// Mitsubishi GX Works2 project: ProjectGroup11   PLC: FX3G

// global labels: Global1
VAR_GLOBAL
  StartSwitch AT X002 : BOOL;
  TC_1 AT TC1 : BOOL;
END_VAR
VAR_GLOBAL CONSTANT
  VALUE : INT := 30;
END_VAR
VAR_GLOBAL
  TS_1 AT TS1 : BOOL;
  Y_005 AT Y005 : BOOL;
  OrangeStock AT D1100 : REAL;
  ClementinesStock AT D1102 : REAL;
  PomeloStock : REAL;
  OrangeWash AT D1106 : REAL;
  ClementinesWash AT D1108 : REAL;
  PomeloWash AT D1110 : REAL;
  SquizeContainer AT D1112 : REAL;
END_VAR
VAR_GLOBAL CONSTANT
  MaxOrangeWash : REAL := 100;
END_VAR
VAR_GLOBAL
  collectionSwitch AT X001 : BOOL;
  collectionInProcess AT Y001 : BOOL;
  squizeSwitch AT X011 : BOOL;
  CC_11 AT CC11 : BOOL;
END_VAR
VAR_GLOBAL CONSTANT
  CS11 : INT := 2;
  const : INT := 2;
END_VAR
VAR_GLOBAL
  CS_11 AT CS11 : BOOL;
  StartDaySwitch AT X010 : BOOL;
END_VAR
VAR_GLOBAL CONSTANT
  MinOranges : REAL;
  PomelaCon : REAL;
  ClementinCon : REAL;
END_VAR
VAR_GLOBAL
  Y_10 AT Y010 : BOOL;
  OffSwitch AT X007 : BOOL;
  TC_7 AT TC7 : BOOL;
END_VAR
VAR_GLOBAL CONSTANT
  ValueOff : INT := 30;
  ValueStart1 : INT := 30;
END_VAR
VAR_GLOBAL
  Y_010 AT Y010 : BOOL;
  M_0 AT M0 : BOOL;
  X_7 AT X007 : BOOL;
  TC_200 AT TC200 : BOOL;
  M_1 AT M1 : BOOL;
  TC_2 AT TC2 : BOOL;
  TS_2 AT TS2 : BOOL;
  M_2 AT M2 : BOOL;
  firstBlink AT M3 : BOOL;
  TC_3 AT TC3 : BOOL;
END_VAR
VAR_GLOBAL CONSTANT
  BlinkingTime : INT := 5;
END_VAR
VAR_GLOBAL
  TS_3 AT TS3 : BOOL;
  Blink2 AT M4 : BOOL;
  Blink1 AT M3 : BOOL;
  TC_4 AT TC4 : BOOL;
  TS_4 AT TS4 : BOOL;
  Blink3 AT M5 : BOOL;
  AllGood AT M6 : BOOL;
  NotGood AT M6 : BOOL;
  StartWashSwitch AT X002 : BOOL;
  Wash1 AT M7 : BOOL;
END_VAR
VAR_GLOBAL CONSTANT
  Ratio : REAL := 2.0;
END_VAR
VAR_GLOBAL
  NumOfOrangeToWash AT D1114 : REAL;
  squize1 AT M8 : BOOL;
  fruitToSquize AT D1116 : REAL;
  switchon AT M1 : BOOL;
  MHelp AT X000 : BOOL;
  Help AT M40 : BOOL;
  Y_6 AT Y006 : BOOL;
  M_35 AT M35 : BOOL;
  JuiceTank AT D1118 : REAL;
  M_9 AT M9 : BOOL;
  TC_5 AT TC5 : BOOL;
END_VAR
VAR_GLOBAL CONSTANT
  SquizeTime : INT := 30;
END_VAR
VAR_GLOBAL
  TS_5 AT TS5 : BOOL;
  Y_2 AT Y002 : BOOL;
  Y_3 AT Y003 : BOOL;
  M_10 AT M10 : BOOL;
  CHECK_QUALIY_STAGE AT X003 : BOOL;
  Output AT D1120 : INT;
END_VAR
VAR_GLOBAL CONSTANT
  UpperBound : REAL := 5.0;
  LowerBound : REAL := 1.0;
END_VAR
VAR_GLOBAL
  M_11 AT M11 : BOOL;
  CHECK_IS_COMPLETE AT Y004 : BOOL;
  M_12 AT M12 : BOOL;
  TC_6 AT TC6 : BOOL;
END_VAR
VAR_GLOBAL CONSTANT
  Value_For_Y4 : INT := 50;
END_VAR
VAR_GLOBAL
  TS_6 AT TS6 : BOOL;
  M_45 AT M45 : BOOL;
  Y_004 AT Y004 : BOOL;
  CC_12 AT CC12 : BOOL;
END_VAR
VAR_GLOBAL CONSTANT
  Checks : INT := 2;
END_VAR
VAR_GLOBAL
  M_13 AT M13 : BOOL;
  NeedAnotherCheck AT M14 : BOOL;
  M_14 AT M14 : BOOL;
  Y_4 AT Y004 : BOOL;
END_VAR
VAR_GLOBAL CONSTANT
  NumOfPush3 : INT := 2;
END_VAR
VAR_GLOBAL
  CS_12 AT CS12 : BOOL;
  JuiceBottles AT D1122 : INT;
  M_15 AT M15 : BOOL;
END_VAR
VAR_GLOBAL CONSTANT
  JuiceBottlesAmount : INT := 15;
END_VAR
VAR_GLOBAL
  X_6 AT X006 : BOOL;
  finalButtles AT D8282 : INT;
END_VAR
VAR_GLOBAL CONSTANT
  noRemainder : INT := 1;
END_VAR
VAR_GLOBAL
  M_16 AT M16 : BOOL;
  M_4 AT M4 : BOOL;
  workersParty AT Y007 : BOOL;
  TC_8 AT TC8 : BOOL;
END_VAR
VAR_GLOBAL CONSTANT
  exactAmount : INT := 50;
END_VAR
VAR_GLOBAL
  TS_8 AT TS8 : BOOL;
  Y_0 AT Y000 : BOOL;
  MODOLO AT D1124 : INT;
  TC_9 AT TC9 : BOOL;
END_VAR
VAR_GLOBAL CONSTANT
  PartyTime : INT := 100;
END_VAR
VAR_GLOBAL
  TS_9 AT TS9 : BOOL;
END_VAR
VAR_GLOBAL CONSTANT
  Reset : REAL;
END_VAR
VAR_GLOBAL
  StorageTank AT D1126 : REAL;
END_VAR
VAR_GLOBAL CONSTANT
  ResetInt : INT;
END_VAR
VAR_GLOBAL
  resetAll AT M17 : BOOL;
  C_11 AT CC11 : BOOL;
  C_12 AT CC12 : BOOL;
  TC_10 AT TC10 : BOOL;
  TS_10 AT TS10 : BOOL;
  M_17 AT M17 : BOOL;
  M_18 AT M18 : BOOL;
  M_19 AT M19 : BOOL;
  goodOrangeAmount AT M20 : BOOL;
  goodClemantinAmount AT M21 : BOOL;
  goodPomeloAmount AT M22 : BOOL;
  M_34 AT M34 : BOOL;
  M_100 AT M100 : BOOL;
  StartingOrange AT D1128 : REAL;
  StartingPomelo AT D1130 : REAL;
  StartingClementine AT D1132 : REAL;
END_VAR
VAR_GLOBAL CONSTANT
  con400 : REAL := 400;
END_VAR
VAR_GLOBAL
  ANALOG AT D8281 : INT;
  Analog_float AT D1134 : REAL;
END_VAR
VAR_GLOBAL CONSTANT
  Mul400 : INT := 400;
END_VAR
VAR_GLOBAL
  M_20 AT M20 : BOOL;
  ThrowAndReset AT M89 : BOOL;
  IntStorageTank AT D1136 : INT;
  intGood AT M30 : BOOL;
  AfterDiv AT M31 : BOOL;
  afterMul AT M32 : BOOL;
  JuiceLeft AT D1138 : INT;
  StorageTankInt AT D1140 : INT;
  TC_14 AT TC14 : BOOL;
END_VAR
VAR_GLOBAL CONSTANT
  SadTime : INT := 30;
END_VAR
VAR_GLOBAL
  TS_14 AT TS14 : BOOL;
  No_LEFT AT M33 : BOOL;
END_VAR
VAR_GLOBAL CONSTANT
  TimeIsOFF : INT := 30;
END_VAR
VAR_GLOBAL
  TC_30 AT TC30 : BOOL;
  TS_30 AT TS30 : BOOL;
END_VAR
VAR_GLOBAL CONSTANT
  con_0 : INT;
  con1 : INT := 1;
END_VAR
VAR_GLOBAL
  NoJuiceRemain AT M40 : BOOL;
END_VAR

// task Task_01 (event TRUE, interval 0, priority 31): POU_01

PROGRAM POU_01
VAR
  OnSwitch : BOOL;
  M_92 : BOOL;
  M_92_A : BOOL;
END_VAR
(* structured ladder/FBD written out as ST: instructions are called as NAME(EN, inputs, outputs); _pN, _eN, _tN stand for wires *)
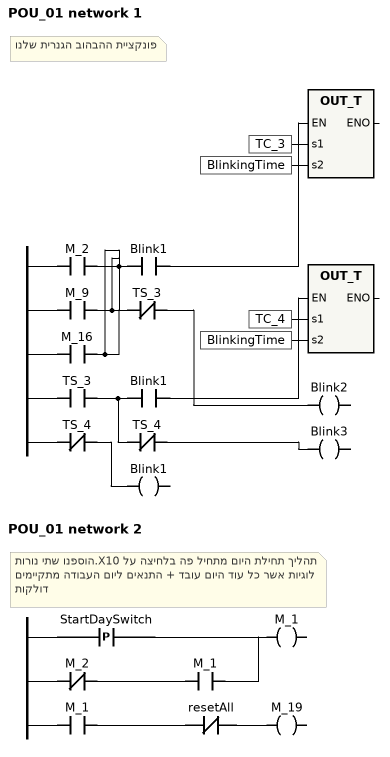
(* network 1 *)
(* פונקציית ההבהוב הגנרית שלנו *)
_p1 := M_2 OR M_9 OR M_16;
OUT_T(_p1 AND Blink1, TC_3, BlinkingTime);
Blink2 := _p1 AND NOT TS_3;
OUT_T(TS_3 AND Blink1, TC_4, BlinkingTime);
Blink3 := TS_3 AND NOT TS_4;
Blink1 := NOT TS_4;
(* network 2 *)
(* תהליך תחילת היום מתחיל פה בלחיצה על X10.הוספנו שתי נורות לוגיות אשר כל עוד היום עובד + התנאים ליום העבודה מתקיימים דולקות *)
M_1 := LDP(TRUE, StartDaySwitch) OR (NOT M_2 AND M_1);
M_19 := M_1 AND NOT resetAll;
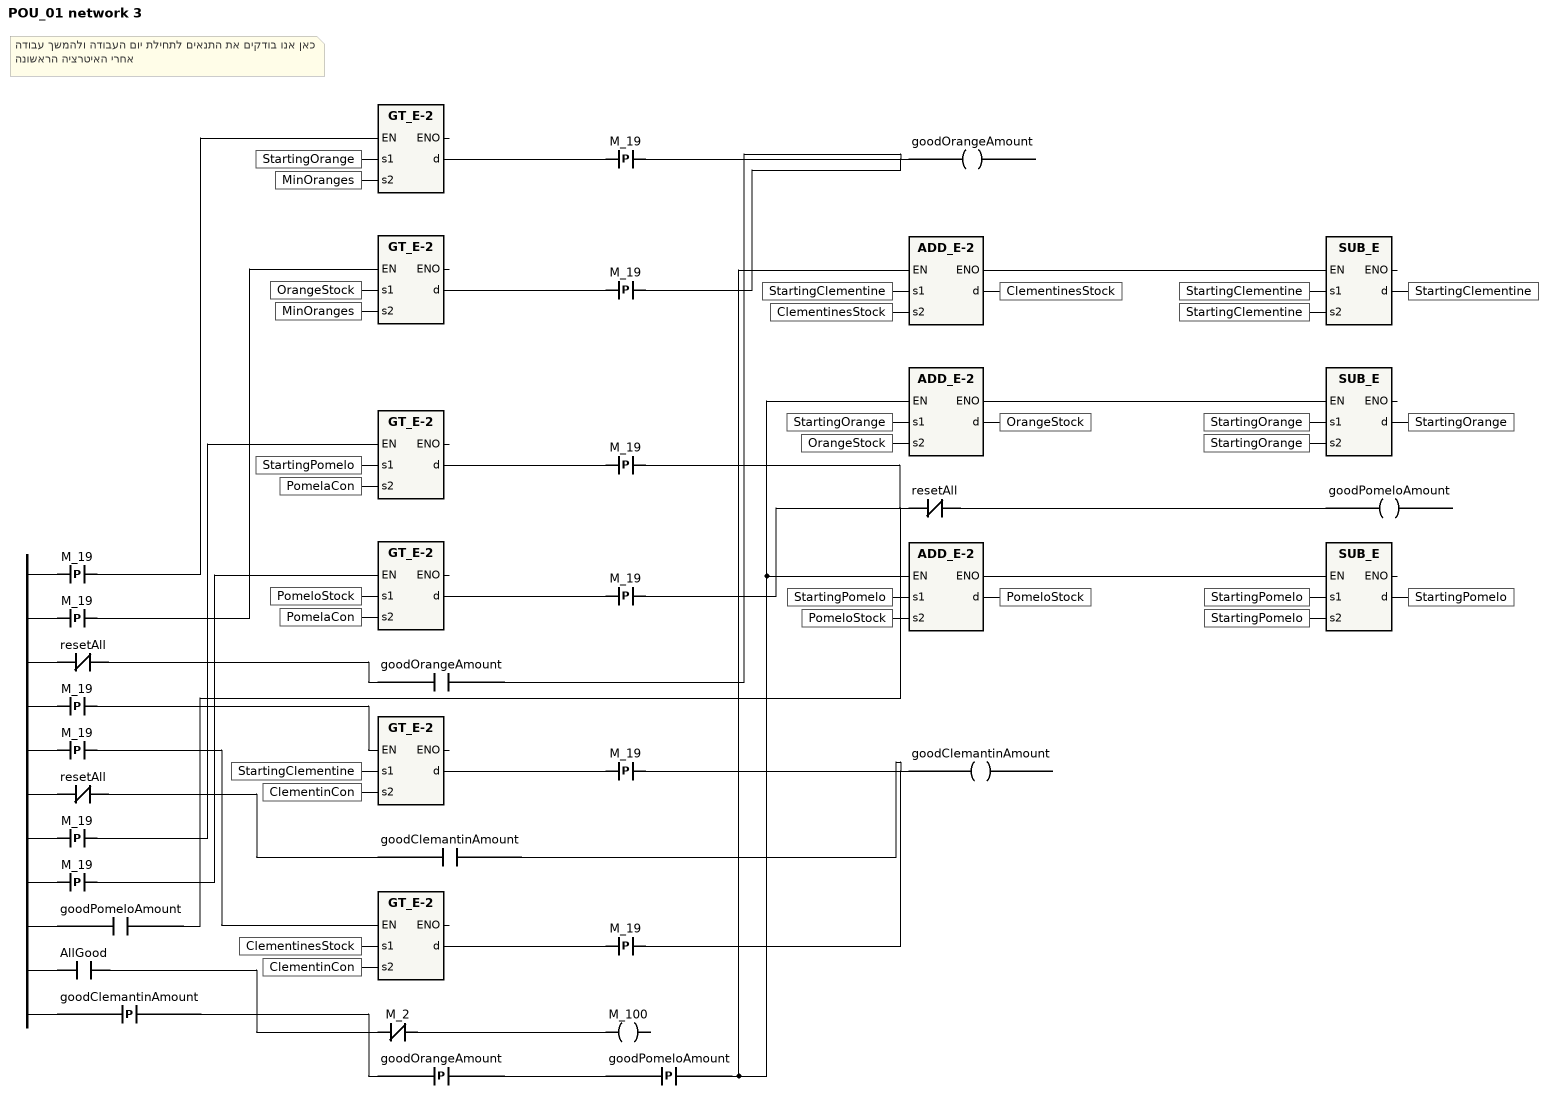
(* network 3 *)
(* כאן אנו בודקים את התנאים לתחילת יום העבודה ולהמשך עבודה אחרי האיטרציה הראשונה *)
GT_E(LDP(TRUE, M_19), StartingOrange, MinOranges, _t1);
GT_E(LDP(TRUE, M_19), OrangeStock, MinOranges, _t2);
goodOrangeAmount := (_t1 AND LDP(TRUE, M_19)) OR (_t2 AND LDP(TRUE, M_19)) OR (NOT resetAll AND goodOrangeAmount);
GT_E(LDP(TRUE, M_19), StartingClementine, ClementinCon, _t3);
GT_E(LDP(TRUE, M_19), ClementinesStock, ClementinCon, _t4);
goodClemantinAmount := (_t3 AND LDP(TRUE, M_19)) OR (_t4 AND LDP(TRUE, M_19)) OR (NOT resetAll AND goodClemantinAmount);
GT_E(LDP(TRUE, M_19), StartingPomelo, PomelaCon, _t5);
GT_E(LDP(TRUE, M_19), PomeloStock, PomelaCon, _t6);
goodPomeloAmount := ((_t5 AND LDP(TRUE, M_19)) OR (_t6 AND LDP(TRUE, M_19)) OR goodPomeloAmount) AND NOT resetAll;
_p7 := LDP(TRUE, goodClemantinAmount) AND LDP(TRUE, goodOrangeAmount) AND LDP(TRUE, goodPomeloAmount);
_e8 := ADD_E(_p7, StartingClementine, ClementinesStock, ClementinesStock);
SUB_E(_e8, StartingClementine, StartingClementine, StartingClementine);
M_100 := AllGood AND NOT M_2;
_e9 := ADD_E(_p7, StartingOrange, OrangeStock, OrangeStock);
SUB_E(_e9, StartingOrange, StartingOrange, StartingOrange);
_e10 := ADD_E(_p7, StartingPomelo, PomeloStock, PomeloStock);
SUB_E(_e10, StartingPomelo, StartingPomelo, StartingPomelo);
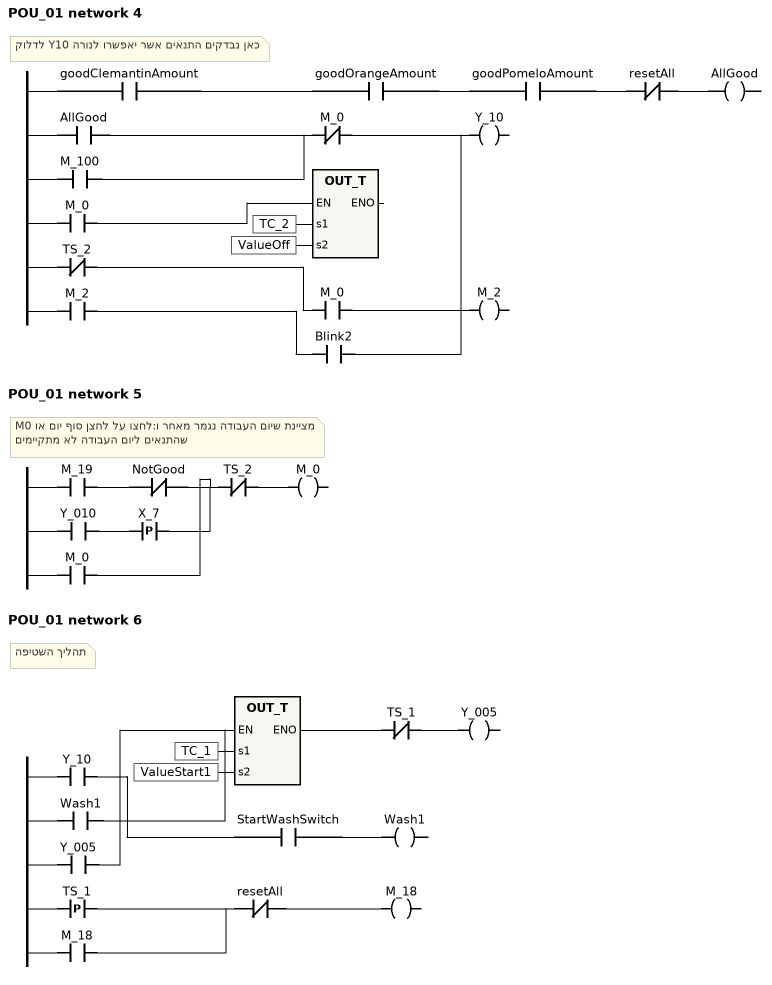
(* network 4 *)
(* כאן נבדקים התנאים אשר יאפשרו לנורה Y10 לדלוק *)
AllGood := goodClemantinAmount AND goodOrangeAmount AND goodPomeloAmount AND NOT resetAll;
Y_10 := ((AllGood OR M_100) AND NOT M_0) OR (M_2 AND Blink2);
OUT_T(M_0, TC_2, ValueOff);
M_2 := NOT TS_2 AND M_0;
(* network 5 *)
(* M0 מציינת שיום העבודה נגמר מאחר ו:לחצו על לחצן סוף יום או שהתנאים ליום העבודה לא מתקיימים *)
M_0 := ((M_19 AND NOT NotGood) OR (Y_010 AND LDP(TRUE, X_7)) OR M_0) AND NOT TS_2;
(* network 6 *)
(* תהליך השטיפה *)
Wash1 := Y_10 AND StartWashSwitch;
_e1 := OUT_T(Wash1 OR Y_005, TC_1, ValueStart1);
Y_005 := _e1 AND NOT TS_1;
M_18 := (LDP(TRUE, TS_1) OR M_18) AND NOT resetAll;
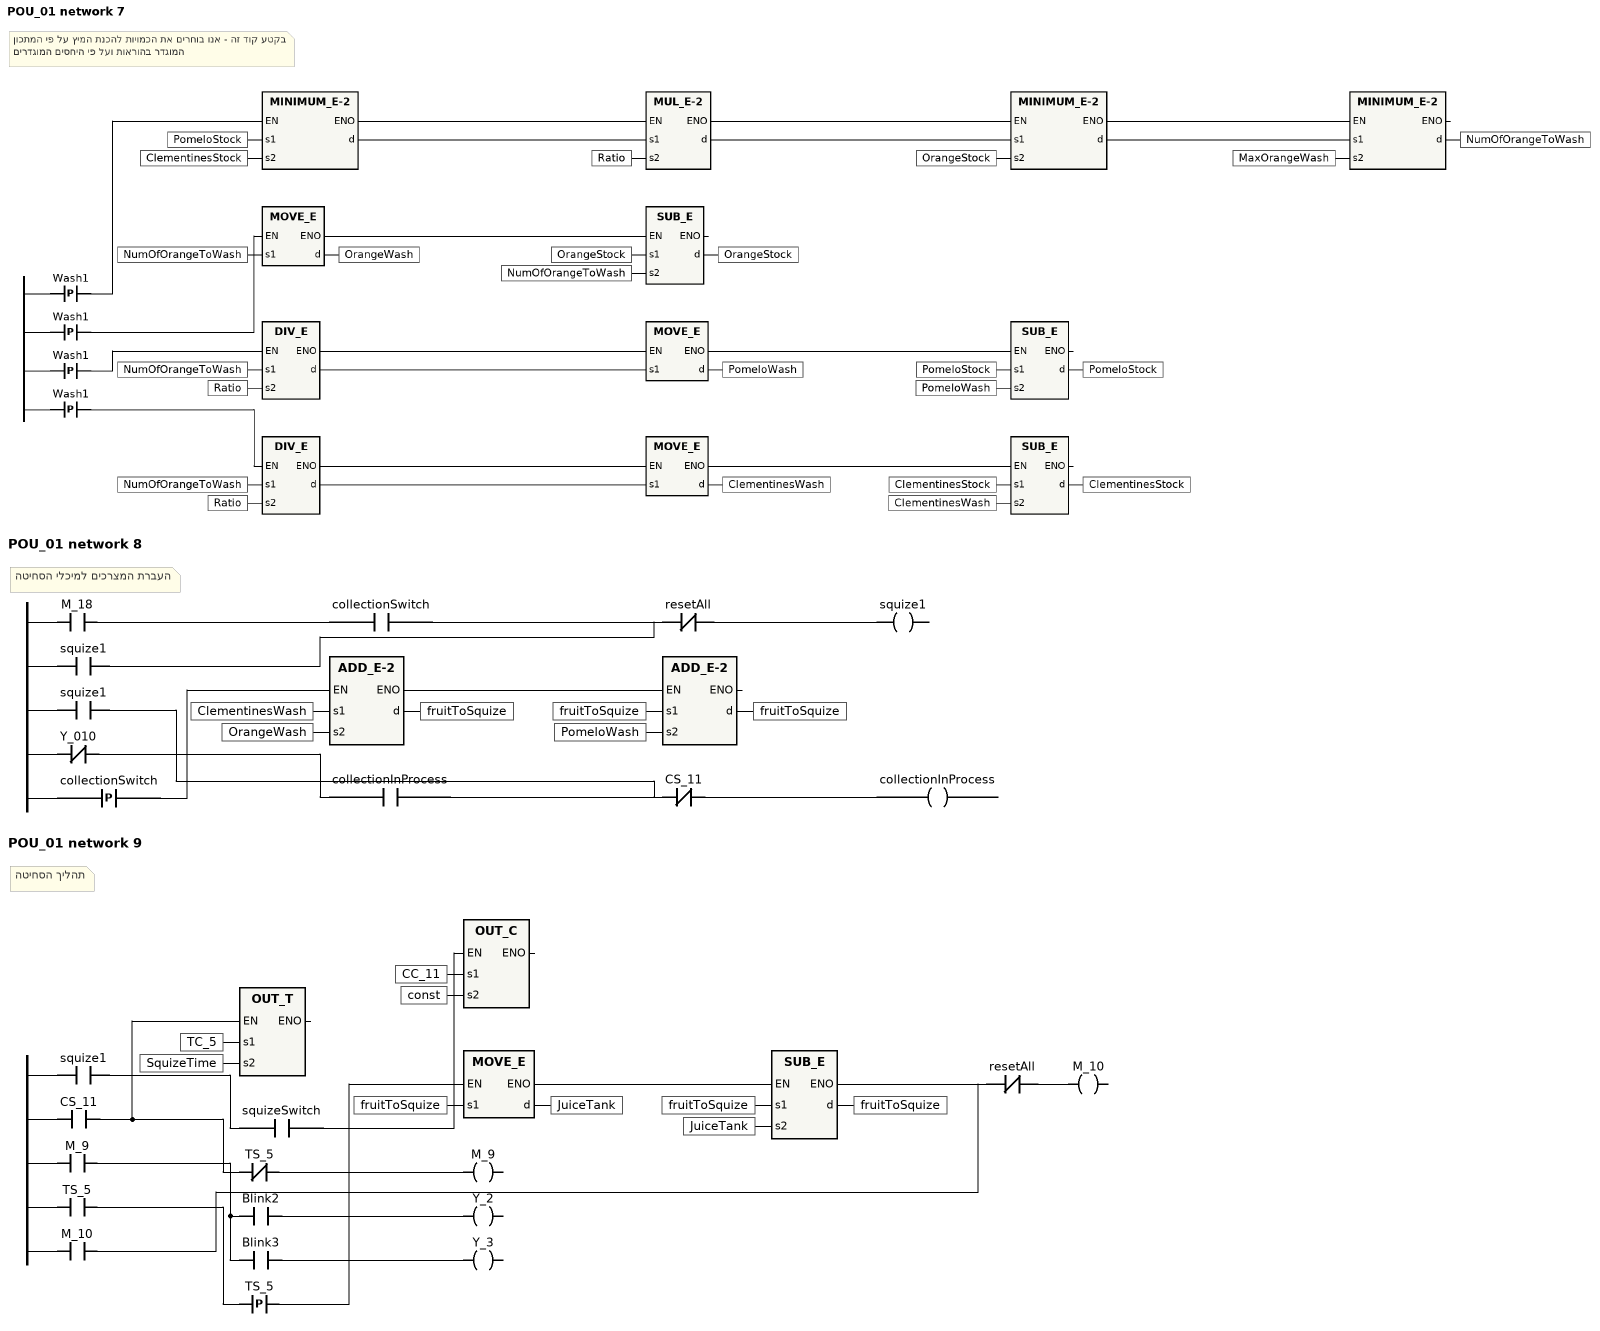
(* network 7 *)
(* בקטע קוד זה - אנו בוחרים את הכמויות להכנת המיץ על פי המתכון המוגדר בהוראות ועל פי היחסים המוגדרים *)
_e2 := MINIMUM_E(LDP(TRUE, Wash1), PomeloStock, ClementinesStock, _t1);
_e4 := MUL_E(_e2, _t1, Ratio, _t3);
_e6 := MINIMUM_E(_e4, _t3, OrangeStock, _t5);
MINIMUM_E(_e6, _t5, MaxOrangeWash, NumOfOrangeToWash);
_e7 := MOVE_E(LDP(TRUE, Wash1), NumOfOrangeToWash, OrangeWash);
SUB_E(_e7, OrangeStock, NumOfOrangeToWash, OrangeStock);
_e9 := DIV_E(LDP(TRUE, Wash1), NumOfOrangeToWash, Ratio, _t8);
_e10 := MOVE_E(_e9, _t8, PomeloWash);
SUB_E(_e10, PomeloStock, PomeloWash, PomeloStock);
_e12 := DIV_E(LDP(TRUE, Wash1), NumOfOrangeToWash, Ratio, _t11);
_e13 := MOVE_E(_e12, _t11, ClementinesWash);
SUB_E(_e13, ClementinesStock, ClementinesWash, ClementinesStock);
(* network 8 *)
(* העברת המצרכים למיכלי הסחיטה *)
squize1 := ((M_18 AND collectionSwitch) OR squize1) AND NOT resetAll;
collectionInProcess := (squize1 OR (NOT Y_010 AND collectionInProcess)) AND NOT CS_11;
_e1 := ADD_E(LDP(TRUE, collectionSwitch), ClementinesWash, OrangeWash, fruitToSquize);
ADD_E(_e1, fruitToSquize, PomeloWash, fruitToSquize);
(* network 9 *)
(* תהליך הסחיטה *)
OUT_C(squize1 AND squizeSwitch, CC_11, const);
OUT_T(CS_11, TC_5, SquizeTime);
M_9 := CS_11 AND NOT TS_5;
Y_2 := M_9 AND Blink2;
Y_3 := M_9 AND Blink3;
_e1 := MOVE_E(TS_5 AND LDP(TRUE, TS_5), fruitToSquize, JuiceTank);
_e2 := SUB_E(_e1, fruitToSquize, JuiceTank, fruitToSquize);
M_10 := (_e2 OR M_10) AND NOT resetAll;
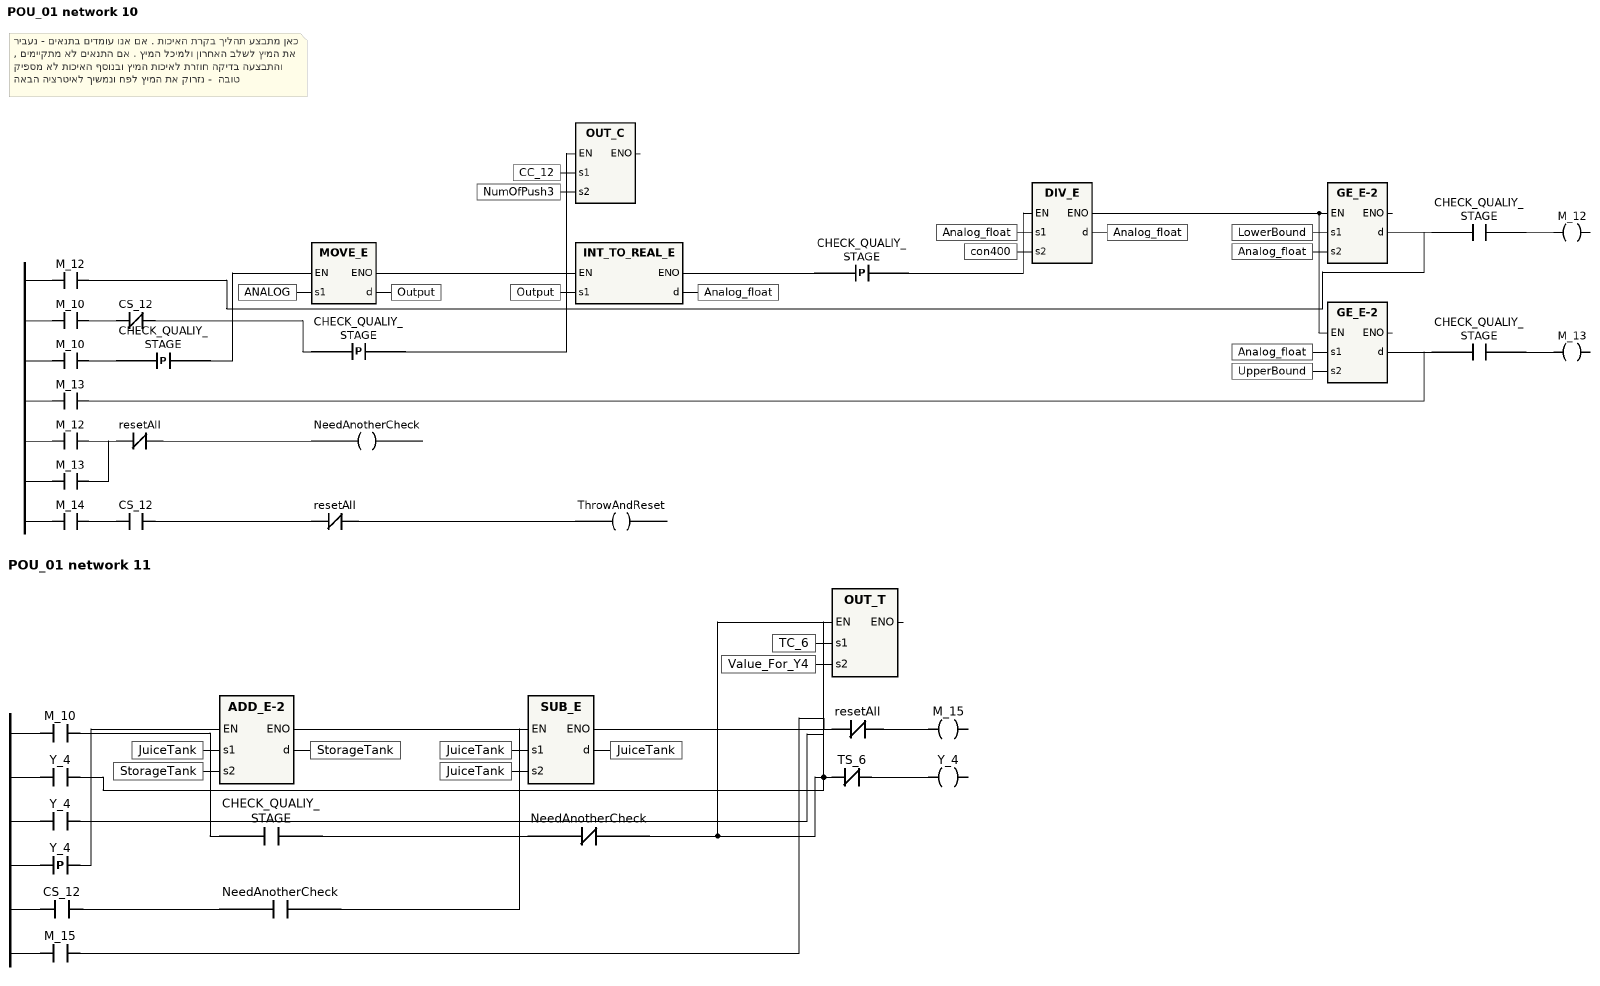
(* network 10 *)
(* כאן מתבצע תהליך בקרת האיכות . אם אנו עומדים בתנאים - נעביר את המיץ לשלב האחרון ולמיכל המיץ . אם התנאים לא מתקיימים , והתבצעה בדיקה חוזרת לאיכות המיץ ובנוסף האיכות לא מספיק טובה  - נזרוק את המיץ לפח ונמשיך לאיטרציה הבאה *)
OUT_C(M_10 AND NOT CS_12 AND LDP(TRUE, CHECK_QUALIY_STAGE), CC_12, NumOfPush3);
_e1 := MOVE_E(M_10 AND LDP(TRUE, CHECK_QUALIY_STAGE), ANALOG, Output);
_e2 := INT_TO_REAL_E(_e1, Output, Analog_float);
_e3 := DIV_E(_e2 AND LDP(TRUE, CHECK_QUALIY_STAGE), Analog_float, con400, Analog_float);
GE_E(_e3, LowerBound, Analog_float, _t4);
M_12 := (M_12 OR _t4) AND CHECK_QUALIY_STAGE;
GE_E(_e3, Analog_float, UpperBound, _t5);
M_13 := (_t5 OR M_13) AND CHECK_QUALIY_STAGE;
NeedAnotherCheck := (M_12 OR M_13) AND NOT resetAll;
ThrowAndReset := M_14 AND CS_12 AND NOT resetAll;
(* network 11 *)
_p1 := (M_10 AND CHECK_QUALIY_STAGE AND NOT NeedAnotherCheck) OR Y_4;
Y_4 := _p1 AND NOT TS_6;
OUT_T(_p1, TC_6, Value_For_Y4);
_e2 := ADD_E(LDP(TRUE, Y_4), JuiceTank, StorageTank, StorageTank);
_e3 := SUB_E(_e2 OR (CS_12 AND NeedAnotherCheck), JuiceTank, JuiceTank, JuiceTank);
M_15 := (Y_4 OR _e3 OR M_15) AND NOT resetAll;
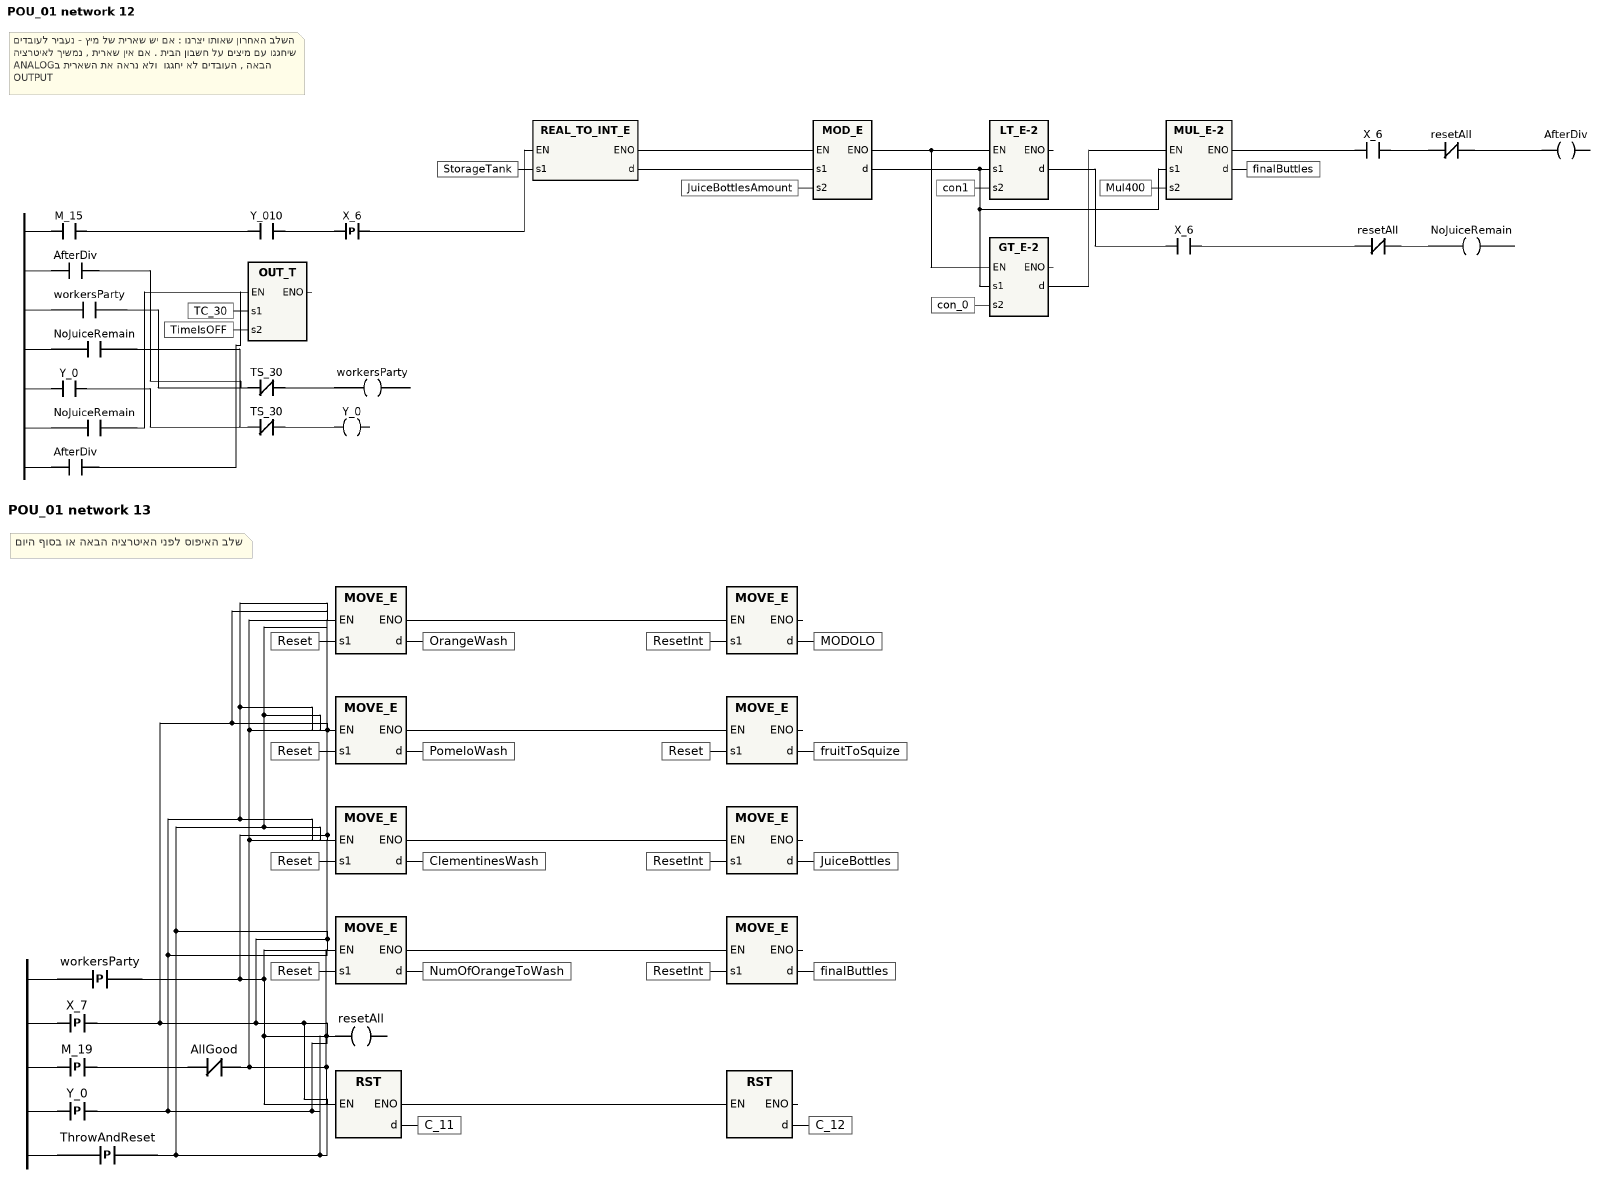
(* network 12 *)
(* השלב האחרון שאותו יצרנו : אם יש שארית של מיץ - נעביר לעובדים שיחגגו עם מיצים על חשבון הבית . אם אין שארית , נמשיך לאיטרציה הבאה , העובדים לא יחגגו  ולא נראה את השארית בANALOG OUTPUT *)
_e2 := REAL_TO_INT_E(M_15 AND Y_010 AND LDP(TRUE, X_6), StorageTank, _t1);
_e4 := MOD_E(_e2, _t1, JuiceBottlesAmount, _t3);
LT_E(_e4, _t3, con1, _t5);
NoJuiceRemain := _t5 AND X_6 AND NOT resetAll;
GT_E(_e4, _t3, con_0, _t6);
_e7 := MUL_E(_t6, _t3, Mul400, finalButtles);
AfterDiv := _e7 AND X_6 AND NOT resetAll;
workersParty := (AfterDiv OR workersParty) AND NOT TS_30;
Y_0 := (NoJuiceRemain OR Y_0) AND NOT TS_30;
OUT_T(NoJuiceRemain OR AfterDiv, TC_30, TimeIsOFF);
(* network 13 *)
(* שלב האיפוס לפני האיטרציה הבאה או בסוף היום *)
_p1 := LDP(TRUE, workersParty) OR LDP(TRUE, X_7) OR (LDP(TRUE, M_19) AND NOT AllGood) OR LDP(TRUE, Y_0) OR LDP(TRUE, ThrowAndReset);
_e2 := MOVE_E(_p1, Reset, OrangeWash);
MOVE_E(_e2, ResetInt, MODOLO);
_e3 := MOVE_E(_p1, Reset, PomeloWash);
MOVE_E(_e3, Reset, fruitToSquize);
_e4 := MOVE_E(_p1, Reset, ClementinesWash);
MOVE_E(_e4, ResetInt, JuiceBottles);
_e5 := MOVE_E(_p1, Reset, NumOfOrangeToWash);
MOVE_E(_e5, ResetInt, finalButtles);
_e6 := RST(_p1, C_11);
RST(_e6, C_12);
resetAll := _p1;
END_PROGRAM
